(* CODESYS project Projektni_zadatak_gotov.project

Project tree, tasks and I/O mapping:
  Device : CECC-S, Festo AG & Co. KG, order no. 574416, version 3.5.7.27
    application Application
      libraries: Standard, * (System); SysTime, 3.5.9.0 (System); SysTypes Interfaces, * (System); Util, * (System)
      task MainTask (cyclic, interval t#20ms, priority 20) calls PLC_PRG
      program PLC_PRG [LD]
      visualisation Visualization_1
    Onboard : CECC 14I/8O, Festo AG & Co. KG, version 3.4.5.5
        unmapped channels: Onboard Input, Onboard Output
      Digital Inputs
          unmapped channels: Onboard Input
      Digital Outputs
          unmapped channels: Onboard Output
  text list GlobalTextList
*)

// Device/Application/PLC_PRG
PROGRAM PLC_PRG
VAR
	S1 : BOOL;
	S2 : BOOL;
	H1 : BOOL;
	H2 : BOOL;
	H3 : BOOL;
	H4 : BOOL;
	V0 : BOOL;
	V1 : BOOL;
	V2 : BOOL;
	V3 : BOOL;
	V4 : BOOL;
	p : TIME;
	POT : INT;
	
	REAL_TIME : RTC;
	
	SEKUNDE :UDINT;
	REZULTAT :UDINT;
	DATUM_VREME :DT; //DATE TIME
	VREME : TOD; //TOD-TIME OF DAY (VREME DANA)
	RADNO_VREME : BOOL;
	RADNO_VREME_VIKEND : BOOL;
	DAN : DATE;
	DAN_U_NEDELJI : UINT;
	
	TAJMER1: TON;
	TAJMER2: TOF;
	TAJMER3: TON;
	TAJMER4: TON;
	TAJMER5: TON;
	TAKT: BOOL := FALSE;
	KORAK : INT := 1;
	REZIM : INT := 1;
	FLAGTON: BOOL;
	FLAGTON1: BOOL;
	PROMENLJIVA : INT;
	REZIM2: BOOL;
	FLAG_KRAJ_R1: BOOL;
	FLAG_KRAJ_R2: BOOL;
	FLAG_GASENJE: BOOL;	
END_VAR
VAR // added by the converter: edge detectors and wires of the graphical bodies
    _w1, _w2, _w3, _w4, _w5, _w6, _w7, _w8, _w9, _w10, _w11, _w12, _w13, _w14, _w15, _w16, _w17, _w18, _w19 : BOOL;
END_VAR

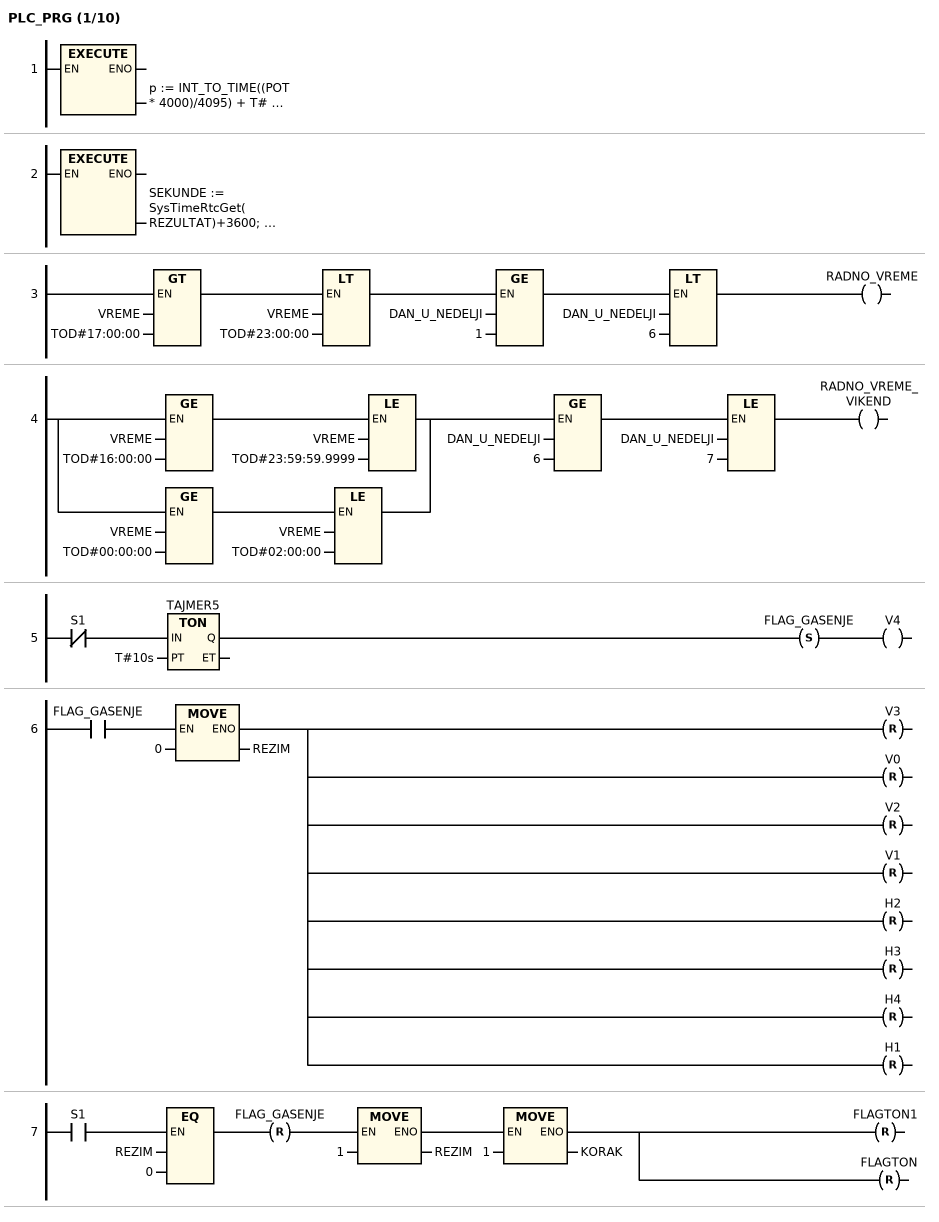
// NETWORK 1
p := INT_TO_TIME((POT * 4000)/4095) + T#1000MS;

// NETWORK 2
SEKUNDE := SysTimeRtcGet(REZULTAT)+3600; //OČITANO TRENUTNO VREME
DATUM_VREME := UDINT_TO_DT(SEKUNDE); //SEKUDNE U DATUM_VREME
VREME := DT_TO_TOD(DATUM_VREME); //KOLIKO JE TRENUTNO SATI
DAN := DT_TO_DATE(DATUM_VREME);
DAN_U_NEDELJI := DWORD_TO_UINT(((DATE_TO_DWORD(DAN)/86400)+3)MOD 7) +1; //KOJI JE DAN U NEDELJI

// NETWORK 3
RADNO_VREME := VREME > (TOD#17:00:00) AND VREME < (TOD#23:00:00) AND DAN_U_NEDELJI >= 1 AND DAN_U_NEDELJI < 6;

// NETWORK 4
RADNO_VREME_VIKEND := (VREME >= (TOD#16:00:00) AND VREME <= (TOD#23:59:59.9999) OR VREME >= (TOD#00:00:00) AND VREME <= (TOD#02:00:00)) AND DAN_U_NEDELJI >= 6 AND DAN_U_NEDELJI <= 7;

// NETWORK 5
TAJMER5(IN := NOT S1, PT := T#10s); // TON
FLAG_GASENJE S= TAJMER5.Q;
V4 := TAJMER5.Q;

// NETWORK 6
_w1 := FLAG_GASENJE;
IF _w1 THEN REZIM := 0; END_IF
V3 R= _w1;
V0 R= _w1;
V2 R= _w1;
V1 R= _w1;
H2 R= _w1;
H3 R= _w1;
H4 R= _w1;
H1 R= _w1;

// NETWORK 7
_w2 := S1 AND REZIM = 0;
FLAG_GASENJE R= _w2;
IF _w2 THEN REZIM := 1; END_IF
IF _w2 THEN KORAK := 1; END_IF
FLAGTON1 R= _w2;
FLAGTON R= _w2;

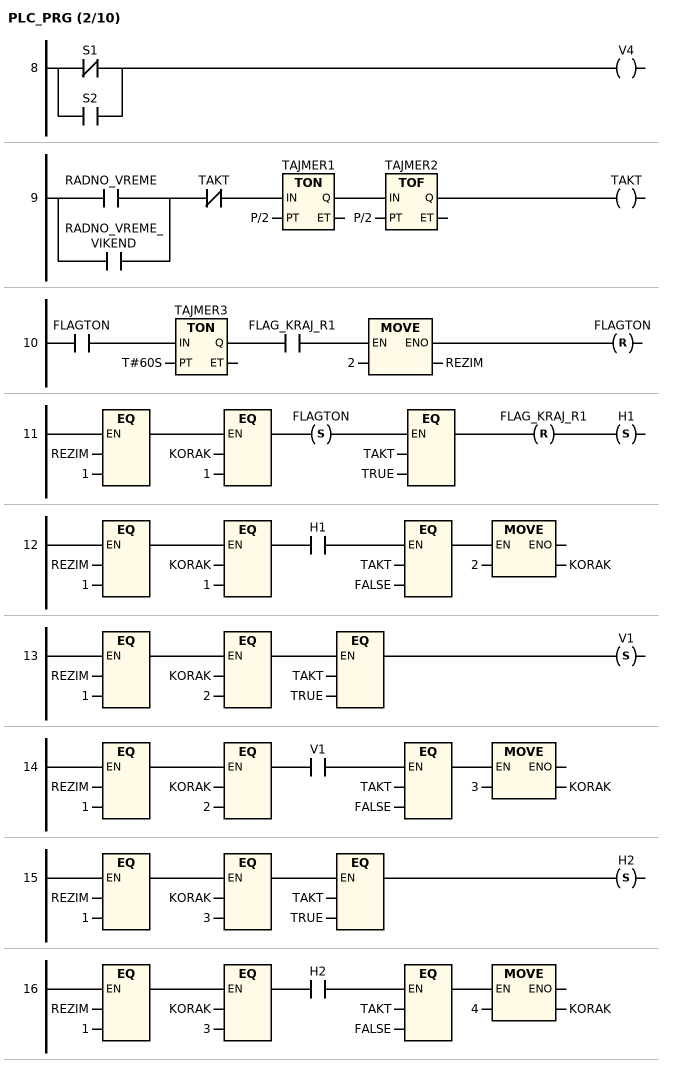
// NETWORK 8
V4 := NOT S1 OR S2;

// NETWORK 9
TAJMER1(IN := (RADNO_VREME OR RADNO_VREME_VIKEND) AND NOT TAKT, PT := P/2); // TON
TAJMER2(IN := TAJMER1.Q, PT := P/2); // TOF
TAKT := TAJMER2.Q;

// NETWORK 10
TAJMER3(IN := FLAGTON, PT := T#60S); // TON
_w3 := TAJMER3.Q AND FLAG_KRAJ_R1;
IF _w3 THEN REZIM := 2; END_IF
FLAGTON R= _w3;

// NETWORK 11
_w4 := REZIM = 1 AND KORAK = 1;
FLAGTON S= _w4;
_w5 := _w4 AND TAKT = TRUE;
FLAG_KRAJ_R1 R= _w5;
H1 S= _w5;

// NETWORK 12
IF (REZIM = 1 AND KORAK = 1) AND H1 AND TAKT = FALSE THEN KORAK := 2; END_IF

// NETWORK 13
V1 S= REZIM = 1 AND KORAK = 2 AND TAKT = TRUE;

// NETWORK 14
IF (REZIM = 1 AND KORAK = 2) AND V1 AND TAKT = FALSE THEN KORAK := 3; END_IF

// NETWORK 15
H2 S= REZIM = 1 AND KORAK = 3 AND TAKT = TRUE;

// NETWORK 16
IF (REZIM = 1 AND KORAK = 3) AND H2 AND TAKT = FALSE THEN KORAK := 4; END_IF

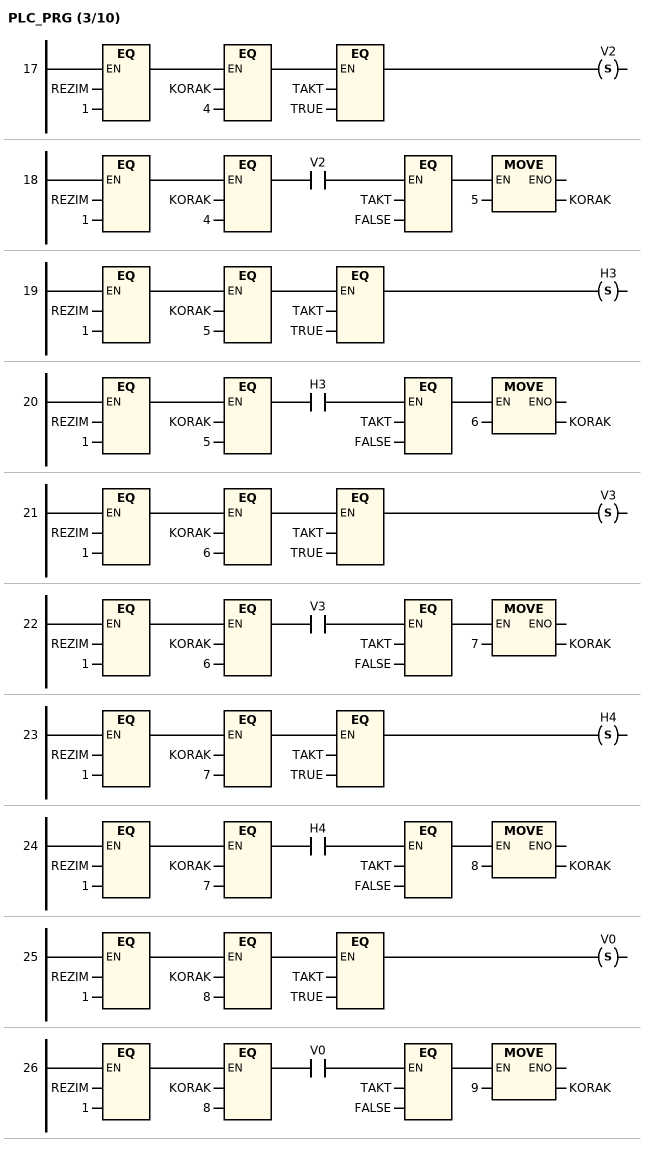
// NETWORK 17
V2 S= REZIM = 1 AND KORAK = 4 AND TAKT = TRUE;

// NETWORK 18
IF (REZIM = 1 AND KORAK = 4) AND V2 AND TAKT = FALSE THEN KORAK := 5; END_IF

// NETWORK 19
H3 S= REZIM = 1 AND KORAK = 5 AND TAKT = TRUE;

// NETWORK 20
IF (REZIM = 1 AND KORAK = 5) AND H3 AND TAKT = FALSE THEN KORAK := 6; END_IF

// NETWORK 21
V3 S= REZIM = 1 AND KORAK = 6 AND TAKT = TRUE;

// NETWORK 22
IF (REZIM = 1 AND KORAK = 6) AND V3 AND TAKT = FALSE THEN KORAK := 7; END_IF

// NETWORK 23
H4 S= REZIM = 1 AND KORAK = 7 AND TAKT = TRUE;

// NETWORK 24
IF (REZIM = 1 AND KORAK = 7) AND H4 AND TAKT = FALSE THEN KORAK := 8; END_IF

// NETWORK 25
V0 S= REZIM = 1 AND KORAK = 8 AND TAKT = TRUE;

// NETWORK 26
IF (REZIM = 1 AND KORAK = 8) AND V0 AND TAKT = FALSE THEN KORAK := 9; END_IF

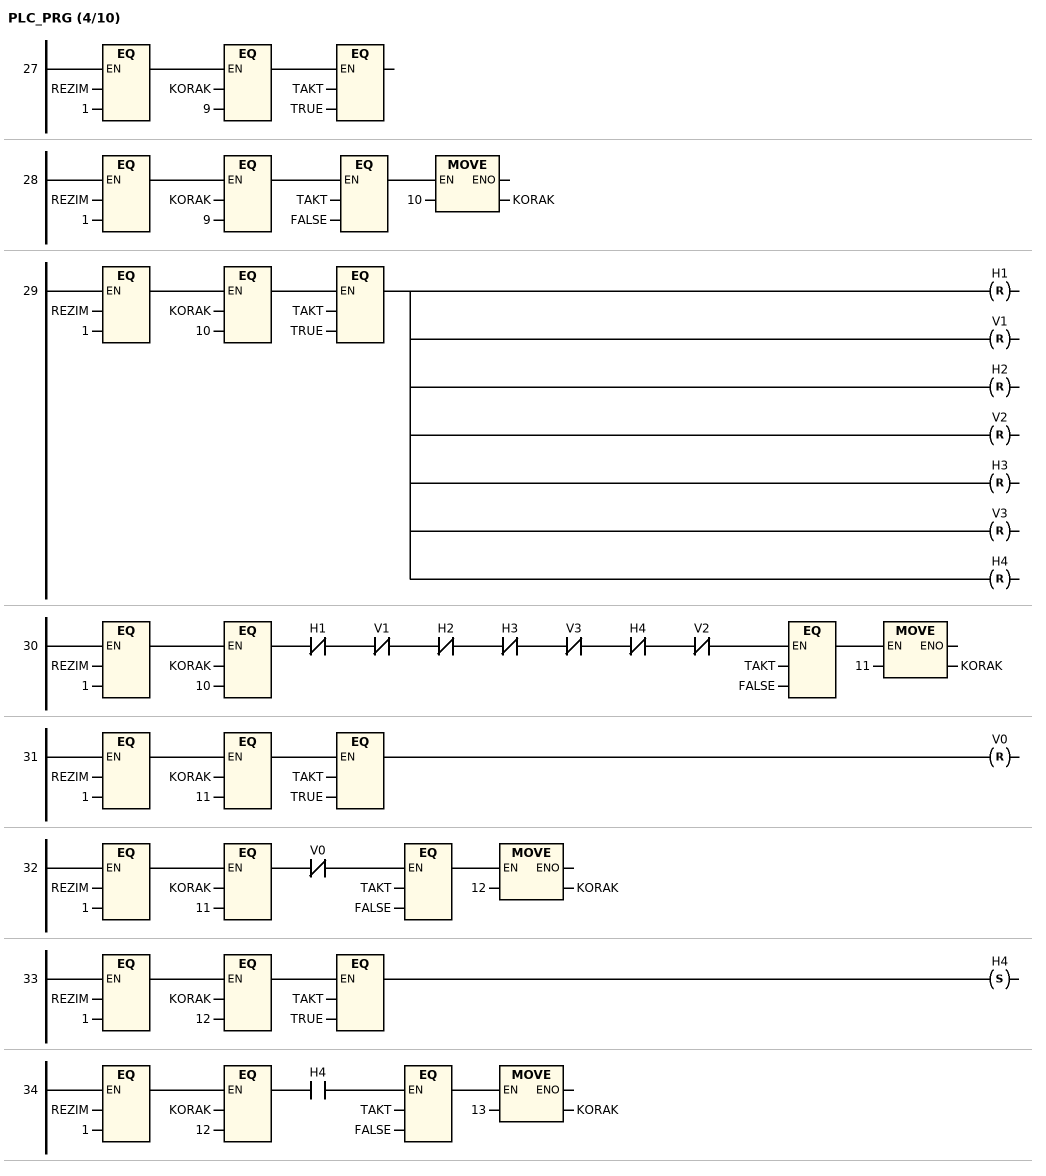
// NETWORK 27
(* REZIM = 1 AND KORAK = 9 AND TAKT = TRUE; result not used *)

// NETWORK 28
IF REZIM = 1 AND KORAK = 9 AND TAKT = FALSE THEN KORAK := 10; END_IF

// NETWORK 29
_w6 := REZIM = 1 AND KORAK = 10 AND TAKT = TRUE;
H1 R= _w6;
V1 R= _w6;
H2 R= _w6;
V2 R= _w6;
H3 R= _w6;
V3 R= _w6;
H4 R= _w6;

// NETWORK 30
IF (REZIM = 1 AND KORAK = 10) AND NOT H1 AND NOT V1 AND NOT H2 AND NOT H3 AND NOT V3 AND NOT H4 AND NOT V2 AND TAKT = FALSE THEN
    KORAK := 11;
END_IF

// NETWORK 31
V0 R= REZIM = 1 AND KORAK = 11 AND TAKT = TRUE;

// NETWORK 32
IF (REZIM = 1 AND KORAK = 11) AND NOT V0 AND TAKT = FALSE THEN KORAK := 12; END_IF

// NETWORK 33
H4 S= REZIM = 1 AND KORAK = 12 AND TAKT = TRUE;

// NETWORK 34
IF (REZIM = 1 AND KORAK = 12) AND H4 AND TAKT = FALSE THEN KORAK := 13; END_IF

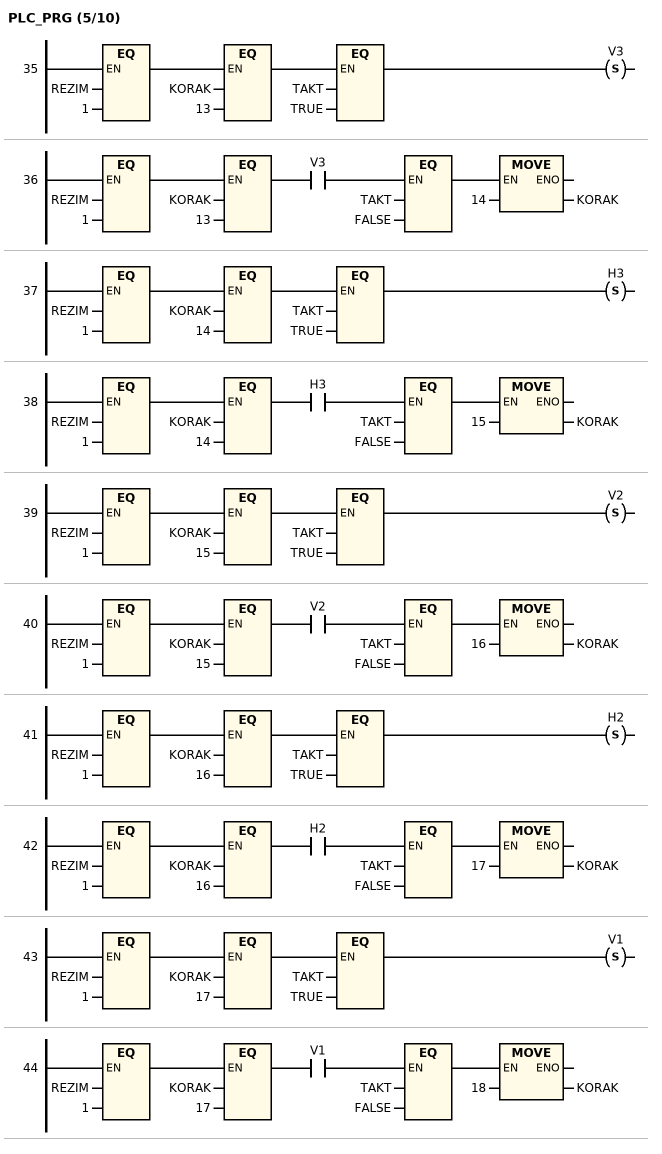
// NETWORK 35
V3 S= REZIM = 1 AND KORAK = 13 AND TAKT = TRUE;

// NETWORK 36
IF (REZIM = 1 AND KORAK = 13) AND V3 AND TAKT = FALSE THEN KORAK := 14; END_IF

// NETWORK 37
H3 S= REZIM = 1 AND KORAK = 14 AND TAKT = TRUE;

// NETWORK 38
IF (REZIM = 1 AND KORAK = 14) AND H3 AND TAKT = FALSE THEN KORAK := 15; END_IF

// NETWORK 39
V2 S= REZIM = 1 AND KORAK = 15 AND TAKT = TRUE;

// NETWORK 40
IF (REZIM = 1 AND KORAK = 15) AND V2 AND TAKT = FALSE THEN KORAK := 16; END_IF

// NETWORK 41
H2 S= REZIM = 1 AND KORAK = 16 AND TAKT = TRUE;

// NETWORK 42
IF (REZIM = 1 AND KORAK = 16) AND H2 AND TAKT = FALSE THEN KORAK := 17; END_IF

// NETWORK 43
V1 S= REZIM = 1 AND KORAK = 17 AND TAKT = TRUE;

// NETWORK 44
IF (REZIM = 1 AND KORAK = 17) AND V1 AND TAKT = FALSE THEN KORAK := 18; END_IF

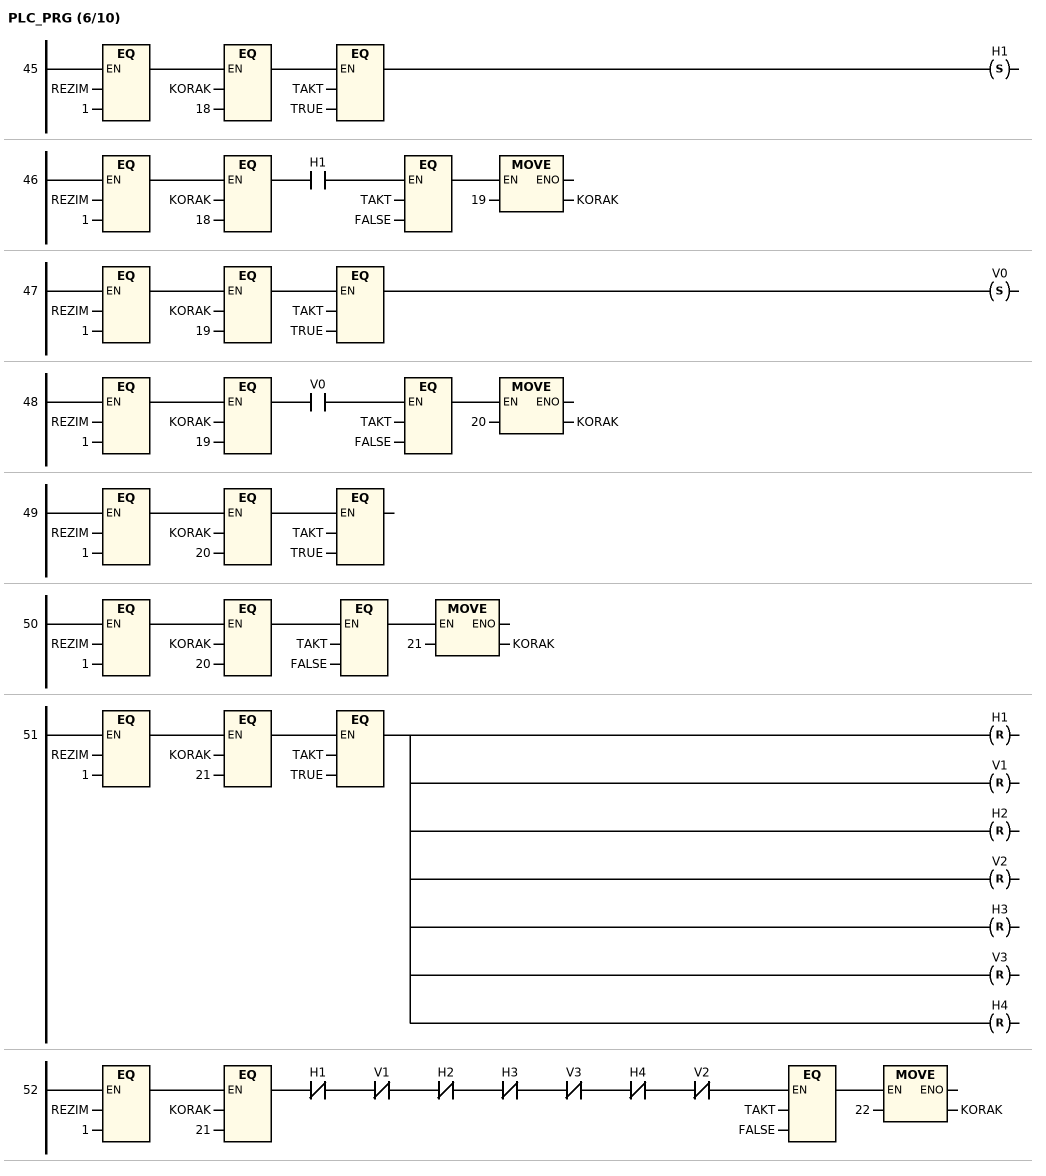
// NETWORK 45
H1 S= REZIM = 1 AND KORAK = 18 AND TAKT = TRUE;

// NETWORK 46
IF (REZIM = 1 AND KORAK = 18) AND H1 AND TAKT = FALSE THEN KORAK := 19; END_IF

// NETWORK 47
V0 S= REZIM = 1 AND KORAK = 19 AND TAKT = TRUE;

// NETWORK 48
IF (REZIM = 1 AND KORAK = 19) AND V0 AND TAKT = FALSE THEN KORAK := 20; END_IF

// NETWORK 49
(* REZIM = 1 AND KORAK = 20 AND TAKT = TRUE; result not used *)

// NETWORK 50
IF REZIM = 1 AND KORAK = 20 AND TAKT = FALSE THEN KORAK := 21; END_IF

// NETWORK 51
_w7 := REZIM = 1 AND KORAK = 21 AND TAKT = TRUE;
H1 R= _w7;
V1 R= _w7;
H2 R= _w7;
V2 R= _w7;
H3 R= _w7;
V3 R= _w7;
H4 R= _w7;

// NETWORK 52
IF (REZIM = 1 AND KORAK = 21) AND NOT H1 AND NOT V1 AND NOT H2 AND NOT H3 AND NOT V3 AND NOT H4 AND NOT V2 AND TAKT = FALSE THEN
    KORAK := 22;
END_IF

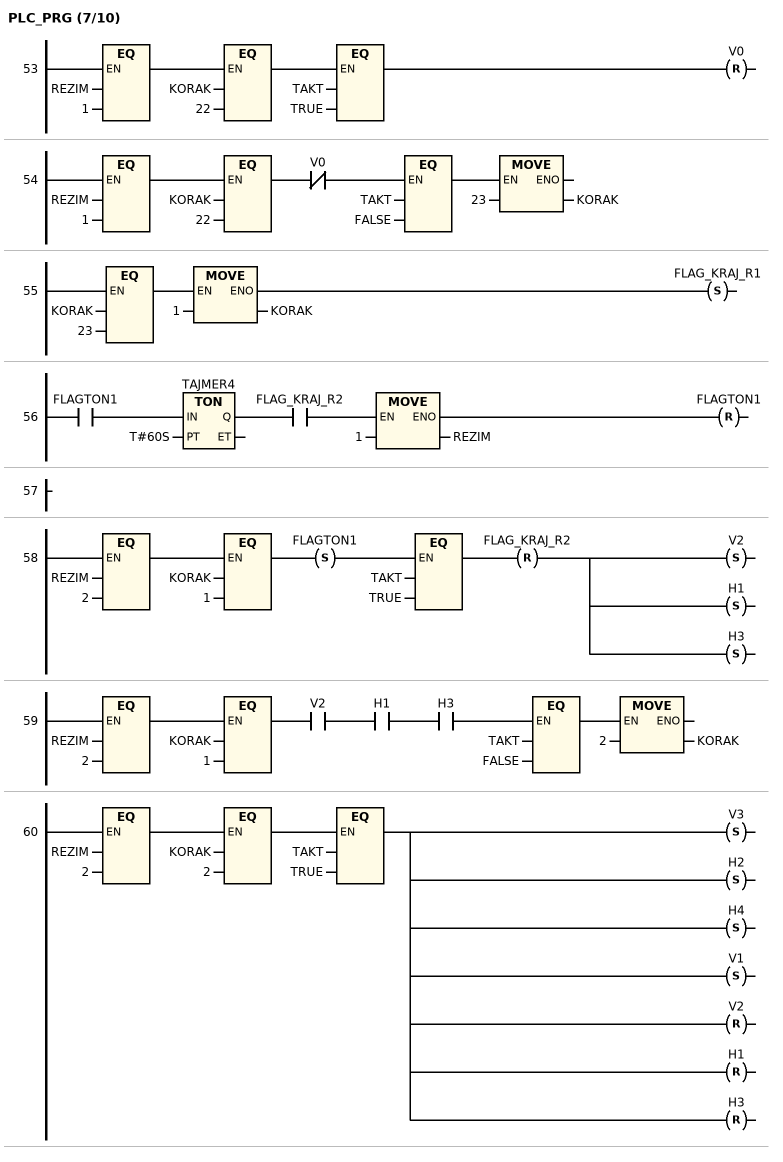
// NETWORK 53
V0 R= REZIM = 1 AND KORAK = 22 AND TAKT = TRUE;

// NETWORK 54
IF (REZIM = 1 AND KORAK = 22) AND NOT V0 AND TAKT = FALSE THEN KORAK := 23; END_IF

// NETWORK 55
_w8 := KORAK = 23;
IF _w8 THEN KORAK := 1; END_IF
FLAG_KRAJ_R1 S= _w8;

// NETWORK 56
TAJMER4(IN := FLAGTON1, PT := T#60S); // TON
_w9 := TAJMER4.Q AND FLAG_KRAJ_R2;
IF _w9 THEN REZIM := 1; END_IF
FLAGTON1 R= _w9;

// NETWORK 57

// NETWORK 58
_w10 := REZIM = 2 AND KORAK = 1;
FLAGTON1 S= _w10;
_w11 := _w10 AND TAKT = TRUE;
FLAG_KRAJ_R2 R= _w11;
V2 S= _w11;
H1 S= _w11;
H3 S= _w11;

// NETWORK 59
IF (REZIM = 2 AND KORAK = 1) AND V2 AND H1 AND H3 AND TAKT = FALSE THEN KORAK := 2; END_IF

// NETWORK 60
_w12 := REZIM = 2 AND KORAK = 2 AND TAKT = TRUE;
V3 S= _w12;
H2 S= _w12;
H4 S= _w12;
V1 S= _w12;
V2 R= _w12;
H1 R= _w12;
H3 R= _w12;

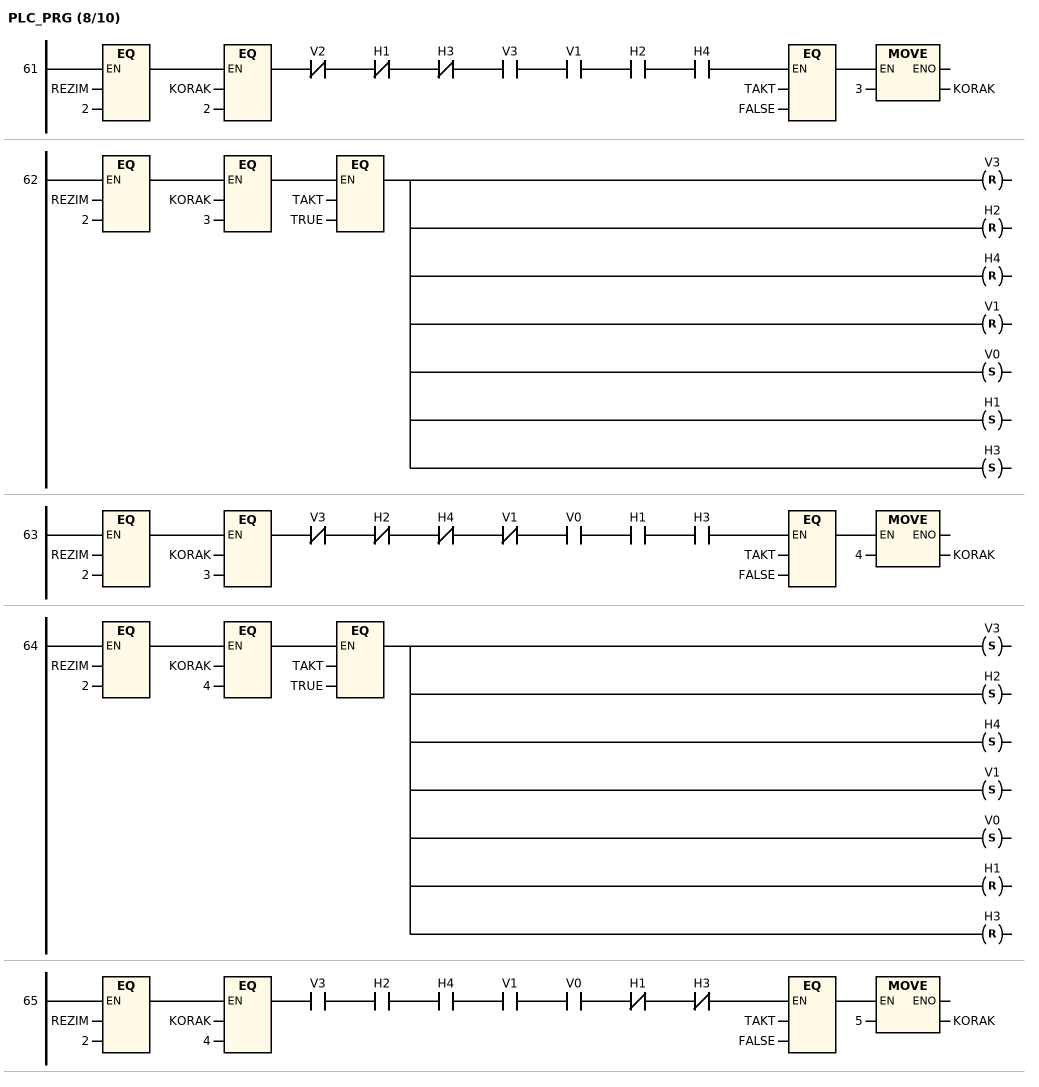
// NETWORK 61
IF (REZIM = 2 AND KORAK = 2) AND NOT V2 AND NOT H1 AND NOT H3 AND V3 AND V1 AND H2 AND H4 AND TAKT = FALSE THEN
    KORAK := 3;
END_IF

// NETWORK 62
_w13 := REZIM = 2 AND KORAK = 3 AND TAKT = TRUE;
V3 R= _w13;
H2 R= _w13;
H4 R= _w13;
V1 R= _w13;
V0 S= _w13;
H1 S= _w13;
H3 S= _w13;

// NETWORK 63
IF (REZIM = 2 AND KORAK = 3) AND NOT V3 AND NOT H2 AND NOT H4 AND NOT V1 AND V0 AND H1 AND H3 AND TAKT = FALSE THEN
    KORAK := 4;
END_IF

// NETWORK 64
_w14 := REZIM = 2 AND KORAK = 4 AND TAKT = TRUE;
V3 S= _w14;
H2 S= _w14;
H4 S= _w14;
V1 S= _w14;
V0 S= _w14;
H1 R= _w14;
H3 R= _w14;

// NETWORK 65
IF (REZIM = 2 AND KORAK = 4) AND V3 AND H2 AND H4 AND V1 AND V0 AND NOT H1 AND NOT H3 AND TAKT = FALSE THEN
    KORAK := 5;
END_IF

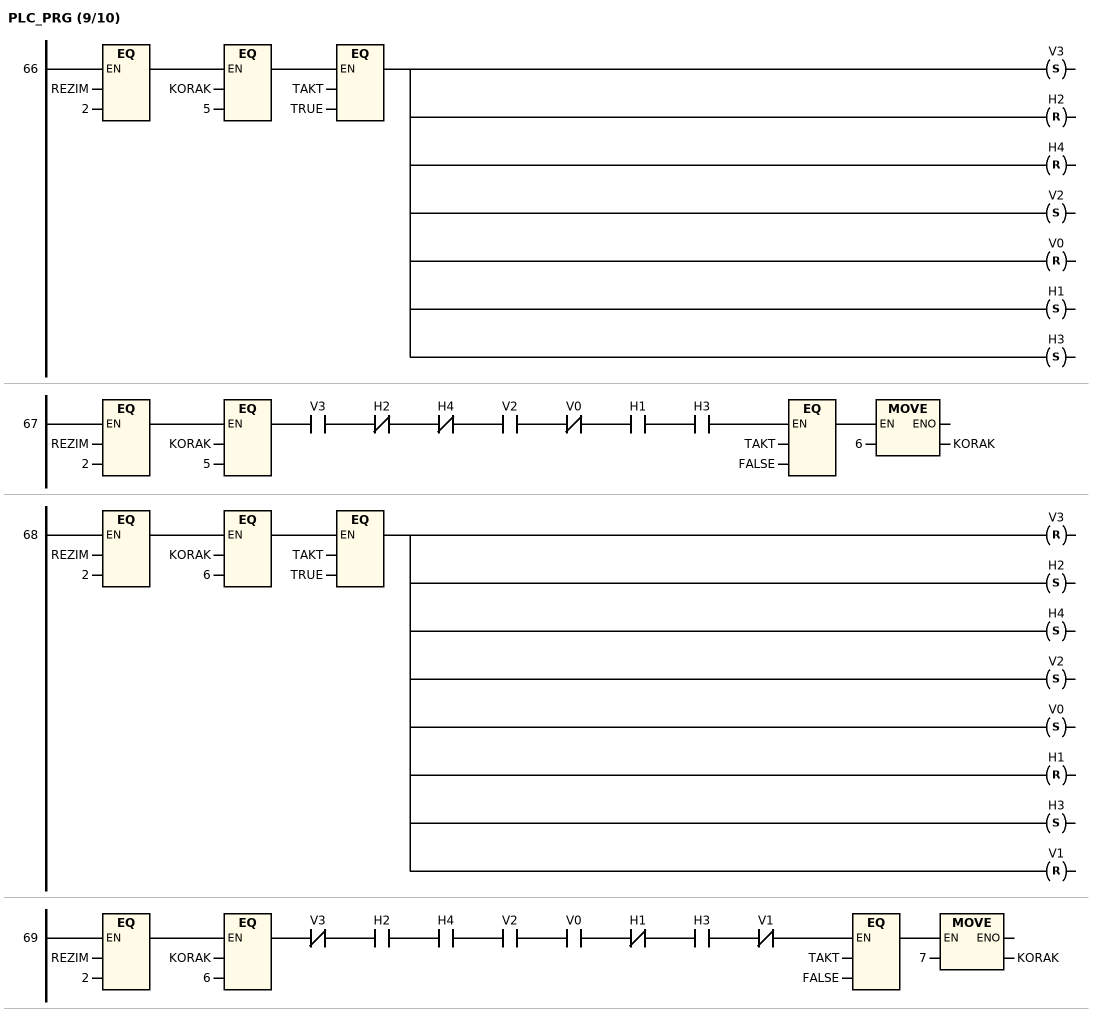
// NETWORK 66
_w15 := REZIM = 2 AND KORAK = 5 AND TAKT = TRUE;
V3 S= _w15;
H2 R= _w15;
H4 R= _w15;
V2 S= _w15;
V0 R= _w15;
H1 S= _w15;
H3 S= _w15;

// NETWORK 67
IF (REZIM = 2 AND KORAK = 5) AND V3 AND NOT H2 AND NOT H4 AND V2 AND NOT V0 AND H1 AND H3 AND TAKT = FALSE THEN
    KORAK := 6;
END_IF

// NETWORK 68
_w16 := REZIM = 2 AND KORAK = 6 AND TAKT = TRUE;
V3 R= _w16;
H2 S= _w16;
H4 S= _w16;
V2 S= _w16;
V0 S= _w16;
H1 R= _w16;
H3 S= _w16;
V1 R= _w16;

// NETWORK 69
IF (REZIM = 2 AND KORAK = 6) AND NOT V3 AND H2 AND H4 AND V2 AND V0 AND NOT H1 AND H3 AND NOT V1 AND TAKT = FALSE THEN
    KORAK := 7;
END_IF

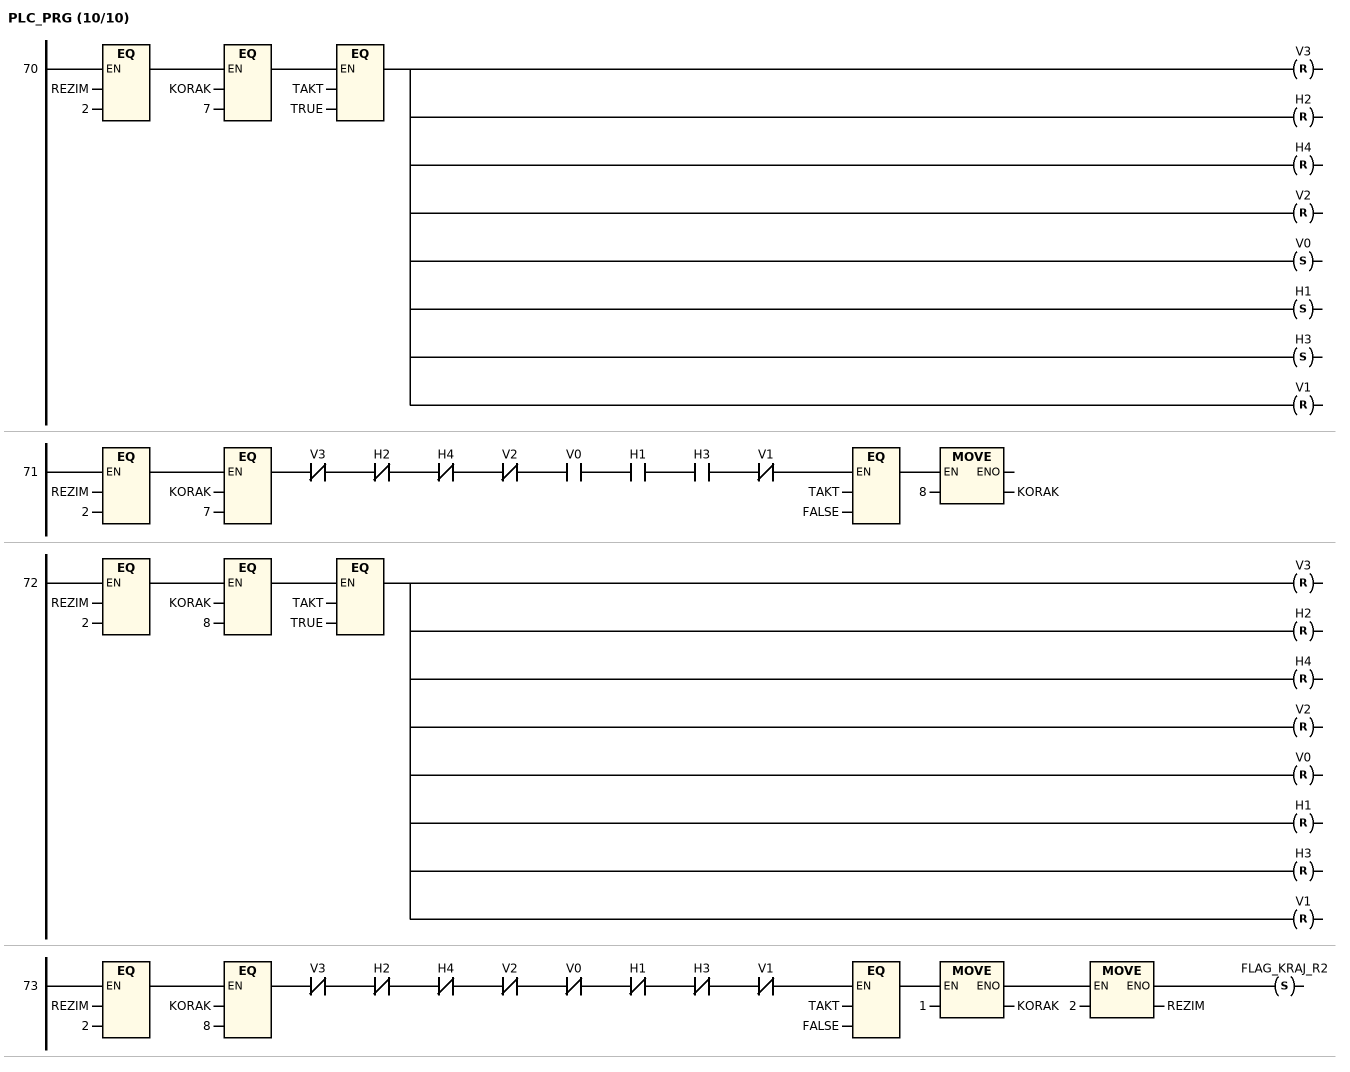
// NETWORK 70
_w17 := REZIM = 2 AND KORAK = 7 AND TAKT = TRUE;
V3 R= _w17;
H2 R= _w17;
H4 R= _w17;
V2 R= _w17;
V0 S= _w17;
H1 S= _w17;
H3 S= _w17;
V1 R= _w17;

// NETWORK 71
IF (REZIM = 2 AND KORAK = 7) AND NOT V3 AND NOT H2 AND NOT H4 AND NOT V2 AND V0 AND H1 AND H3 AND NOT V1 AND TAKT = FALSE THEN
    KORAK := 8;
END_IF

// NETWORK 72
_w18 := REZIM = 2 AND KORAK = 8 AND TAKT = TRUE;
V3 R= _w18;
H2 R= _w18;
H4 R= _w18;
V2 R= _w18;
V0 R= _w18;
H1 R= _w18;
H3 R= _w18;
V1 R= _w18;

// NETWORK 73
_w19 := (REZIM = 2 AND KORAK = 8) AND NOT V3 AND NOT H2 AND NOT H4 AND NOT V2 AND NOT V0 AND NOT H1 AND NOT H3 AND NOT V1 AND TAKT = FALSE;
IF _w19 THEN KORAK := 1; END_IF
IF _w19 THEN REZIM := 2; END_IF
FLAG_KRAJ_R2 S= _w19;

END_PROGRAM

// Device/Application/Visualization_1
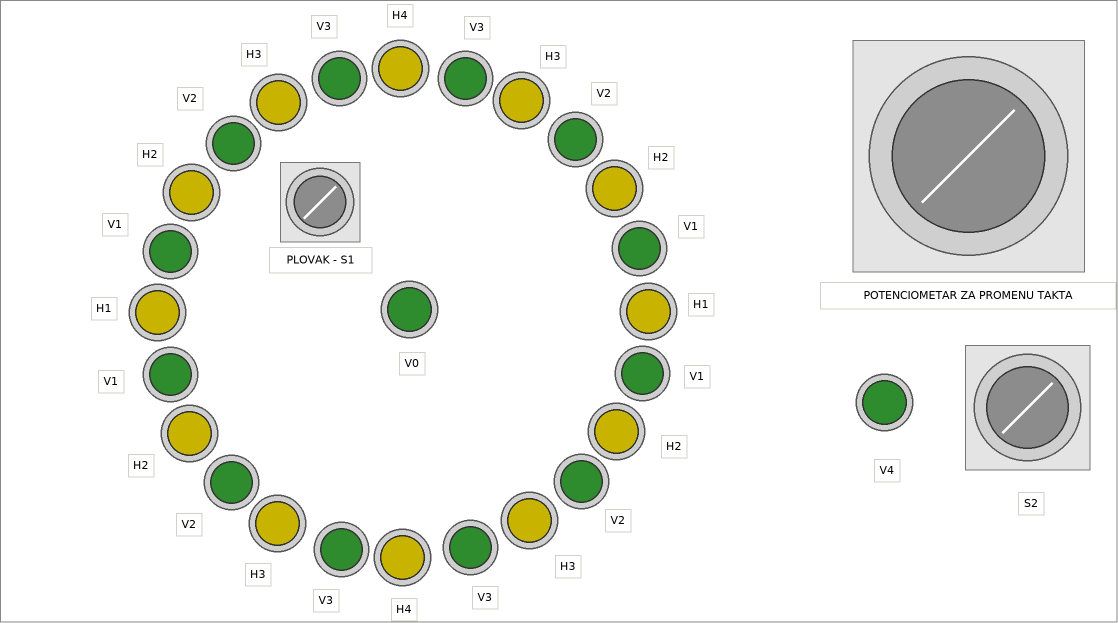
VISUALIZATION Visualization_1  // 1118x623
    Potentiometer360 (845,40 247x232), variable: PLC_PRG.POT, style: Potentiometer-Potentiometer360-Gray, scale format: %d, scale 0..4095
        p2431819421: Outside
    Lamp1 (368,524 69x67), variable: PLC_PRG.H4, style: Lamp-Lamp1-Yellow
    RotarySwitch (965,345 125x125), variable: PLC_PRG.S2, behaviour: TOGGLE, style: Switch-RotarySwitch-Gray
    Lamp1 (850,369 69x67), variable: PLC_PRG.V4, style: Lamp-Lamp1-Green
    Lamp1 (305,517 73x65), variable: PLC_PRG.V3, style: Lamp-Lamp1-Green
    Lamp1 (375,276 69x67), variable: PLC_PRG.V0, style: Lamp-Lamp1-Green
    RotarySwitch (280,162 80x80), variable: PLC_PRG.S1, behaviour: TOGGLE, style: Switch-RotarySwitch-Gray
    Lamp1 (366,35 69x67), variable: PLC_PRG.H4, style: Lamp-Lamp1-Yellow
    Lamp1 (434,515 73x65), variable: PLC_PRG.V3, style: Lamp-Lamp1-Green
    Lamp1 (614,278 69x67), variable: PLC_PRG.H1, style: Lamp-Lamp1-Yellow
    Lamp1 (123,279 69x67), variable: PLC_PRG.H1, style: Lamp-Lamp1-Yellow
    Lamp1 (603,216 73x65), variable: PLC_PRG.V1, style: Lamp-Lamp1-Green
    Lamp1 (606,341 73x65), variable: PLC_PRG.V1, style: Lamp-Lamp1-Green
    Lamp1 (134,342 73x65), variable: PLC_PRG.V1, style: Lamp-Lamp1-Green
    Lamp1 (134,219 73x65), variable: PLC_PRG.V1, style: Lamp-Lamp1-Green
    Lamp1 (303,46 73x65), variable: PLC_PRG.V3, style: Lamp-Lamp1-Green
    Lamp1 (429,46 73x65), variable: PLC_PRG.V3, style: Lamp-Lamp1-Green
    Lamp1 (487,67 69x67), variable: PLC_PRG.H3, style: Lamp-Lamp1-Yellow
    Lamp1 (244,69 69x67), variable: PLC_PRG.H3, style: Lamp-Lamp1-Yellow
    Lamp1 (582,398 69x67), variable: PLC_PRG.H2, style: Lamp-Lamp1-Yellow
    Lamp1 (580,155 69x67), variable: PLC_PRG.H2, style: Lamp-Lamp1-Yellow
    Lamp1 (157,159 69x67), variable: PLC_PRG.H2, style: Lamp-Lamp1-Yellow
    Lamp1 (155,400 69x67), variable: PLC_PRG.H2, style: Lamp-Lamp1-Yellow
    Lamp1 (495,487 69x67), variable: PLC_PRG.H3, style: Lamp-Lamp1-Yellow
    Lamp1 (243,490 69x67), variable: PLC_PRG.H3, style: Lamp-Lamp1-Yellow
    Lamp1 (195,450 73x65), variable: PLC_PRG.V2, style: Lamp-Lamp1-Green
    Lamp1 (197,111 73x65), variable: PLC_PRG.V2, style: Lamp-Lamp1-Green
    Lamp1 (545,449 73x65), variable: PLC_PRG.V2, style: Lamp-Lamp1-Green
    Lamp1 (539,107 73x65), variable: PLC_PRG.V2, style: Lamp-Lamp1-Green
    Textfield (387,4 26x23), "H4"
    Textfield (391,598 26x23), "H4"
    Textfield (688,293 26x23), "H1"
    Textfield (91,297 26x23), "H1"
    Textfield (648,146 26x23), "H2"
    Textfield (661,435 26x23), "H2"
    Textfield (128,454 26x23), "H2"
    Textfield (137,143 26x23), "H2"
    Textfield (540,45 26x23), "H3"
    Textfield (241,43 26x23), "H3"
    Textfield (245,563 26x23), "H3"
    Textfield (555,555 26x23), "H3"
    Textfield (464,16 26x23), "V3"
    Textfield (311,15 26x23), "V3"
    Textfield (472,586 26x23), "V3"
    Textfield (313,589 26x23), "V3"
    Textfield (591,82 26x23), "V2"
    Textfield (177,87 26x23), "V2"
    Textfield (605,509 26x23), "V2"
    Textfield (176,513 26x23), "V2"
    Textfield (102,213 26x23), "V1"
    Textfield (98,370 26x23), "V1"
    Textfield (678,215 26x23), "V1"
    Textfield (684,365 26x23), "V1"
    Textfield (269,247 103x26), "PLOVAK - S1"
    Textfield (399,352 26x23), "V0"
    Textfield (874,459 26x23), "V4"
    Textfield (1018,492 26x23), "S2"
    Textfield (820,282 296x27), "POTENCIOMETAR ZA PROMENU TAKTA"
END_VISUALIZATION
